PROGRAM PRG_TEST
VAR
	fbAnalog2Real_TEST :FB_Raw2Analog_Test;
END_VAR

 TcUnit.RUN();

END_PROGRAM

(* stored: Version 1.1.0.1, ProductVersion 3.1.4024.12
   POU PRG_TEST: Id {ac77a46f-3b28-4b78-ac32-013a1793b016}, SpecialFunc None *)
